ABB RobotStudio station: Solution1.rsstn

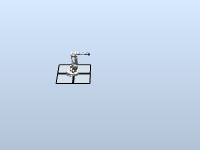
Station Solution1 (saved by RobotStudio 6.8.8148.134)
Controller IRB_2400_12kg_1.55m
  mechanical unit ROB_1: IRB2400_10_150__02, 6 joints, base frame (0, 0, 0) mm
Layout (positions relative to the parent item):
  - IRB2400_10_150__02 [mechanism, from Robots\IRB2400_10_150_G_02.rslib] at (0, 0, 0) mm; joint values [0, 0, 0, 0, 0.5236, 0] (rad or m)
